(* CoDeSys 2.3.9.50 project: 5A.pr6 *)
(* Libraries: STANDARD.LB6 5.6.98 12:03:02 *)

(* POU MAIN, LD *)
PROGRAM MAIN
VAR
	Input AT %IX0.0: BOOL;
	Start AT %IX0.1: BOOL;
	Reject AT %IX0.3: BOOL;
	MainConveyer AT %QX0.0: BOOL;
	Inspection AT %IX0.2: BOOL;
	Divertedgate AT %QX0.1: BOOL;
	B AT %IX0.6: BOOL;
	A: INT;
	C1: CTU;
	C2: CTU;
END_VAR
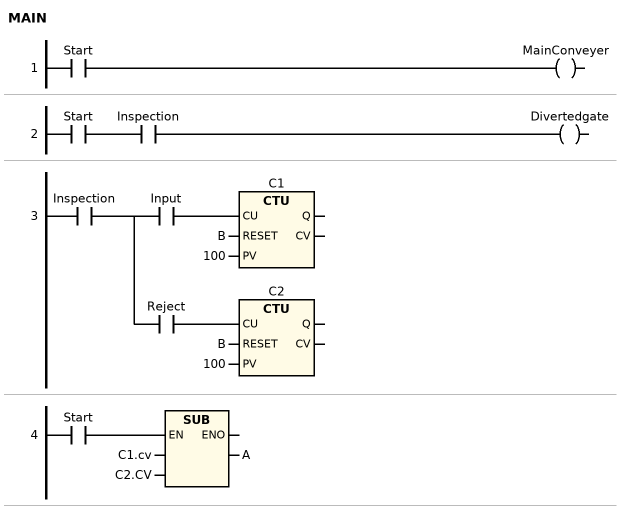
_LD_ (* Ladder Diagram *)
NETWORK 1
	[Start] --- (MainConveyer)
NETWORK 2
	[Start] - [Inspection] --- (Divertedgate)
NETWORK 3
	[Inspection] - { [Input] - C1:CTU(CU: *, RESET: B, PV: 100) | [Reject] - C2:CTU(CU: *, RESET: B, PV: 100) }
NETWORK 4
	[Start]
		EN --- SUB(C1.cv, C2.CV) => A
_END_LD_
(* the same logic as Structured Text *)
(* Network 1 *)
MainConveyer := Start;
(* Network 2 *)
Divertedgate := Start AND Inspection;
(* Network 3 *)
C1(CU := Inspection AND Input, RESET := B, PV := 100);
C2(CU := Inspection AND Reject, RESET := B, PV := 100);
(* Network 4 *)
IF Start THEN
	A := C1.cv - C2.CV;
END_IF;
END_PROGRAM
